TYPE CmpCore :
STRUCT
	
	Framework: Framework;

END_STRUCT
END_TYPE

(* stored: Version 1.1.0.1, ProductVersion 3.1.4024.6
   DUT CmpCore: Id {17db1a67-a561-460c-a797-793fdb2daa5c} *)
